AssertEquals_LREAL(
    Expected := 30.0,
    Actual := fbQ1.GetNormSq(),
    Delta := 1e-10,
    Message := 'Norm squared was not the expected value.'
);

AssertEquals_LREAL(
    Expected := 0.047543581616482,
    Actual := fbQ1.GetNormSq(),
    Delta := 1e-10,
    Message := 'Norm squared was not the expected value.'
);

TEST_FINISHED();
END_METHOD


METHOD PRIVATE TestMakeConjExpectCorrectResult
VAR
    fbQ1 : FB_Quaternion;
END_VAR

TEST('TestMakeConjExpectCorrectResult');

fbQ1.Set(1, 2, 3, 4);
fbQ1.MakeConj();

AssertEquals_LREAL(
    Expected := 1,
    Actual := fbQ1.w,
    Delta := 0.0,
    Message := 'Quaternion 1 [w] was not the expected value.'
);

AssertEquals_LREAL(
    Expected := -2,
    Actual := fbQ1.x,
    Delta := 0.0,
    Message := 'Quaternion 1 [x] was not the expected value.'
);

AssertEquals_LREAL(
    Expected := -3,
    Actual := fbQ1.y,
    Delta := 0.0,
    Message := 'Quaternion 1 [y] was not the expected value.'
);

AssertEquals_LREAL(
    Expected := -4,
    Actual := fbQ1.z,
    Delta := 0.0,
    Message := 'Quaternion 1 [z] was not the expected value.'
);

TEST_FINISHED();
END_METHOD


METHOD PRIVATE TestMulQuatExpectCorrectResult
VAR
    fbQ1 : FB_Quaternion;
    fbQ2 : FB_Quaternion;
    fbQ3 : FB_Quaternion;
END_VAR

TEST('TestMulQuatExpectCorrectResult');

fbQ1.Set(1, 2, 3, 4);
fbQ2.Set(0.217115689381933, -0.00950871632329635, 0.01743264659271, -0.00316957210776545);
fbQ3.Set(2, -1, -5, 2);

fbQ1.MulQuat(fbQ2);
fbQ3.MulQuat(fbQ1);

// Q1
AssertEquals_LREAL(
    Expected := 0.196513470681458,
    Actual := fbQ1.w,
    Delta := 1e-10,
    Message := 'Quaternion 1 [w] was not the expected value.'
);

AssertEquals_LREAL(
    Expected := 0.345483359746434,
    Actual := fbQ1.x,
    Delta := 1e-10,
    Message := 'Quaternion 1 [x] was not the expected value.'
);

AssertEquals_LREAL(
    Expected := 0.637083993660856,
    Actual := fbQ1.y,
    Delta := 1e-10,
    Message := 'Quaternion 1 [y] was not the expected value.'
);

AssertEquals_LREAL(
    Expected := 0.928684627575277,
    Actual := fbQ1.z,
    Delta := 1e-10,
    Message := 'Quaternion 1 [z] was not the expected value.'
);

// Q2
AssertEquals_LREAL(
    Expected := 0.217115689381933,
    Actual := fbQ2.w,
    Delta := 0.0,
    Message := 'Quaternion 2 [w] was not the expected value.'
);

AssertEquals_LREAL(
    Expected := -0.00950871632329635,
    Actual := fbQ2.x,
    Delta := 0.0,
    Message := 'Quaternion 2 [x] was not the expected value.'
);

AssertEquals_LREAL(
    Expected := 0.01743264659271,
    Actual := fbQ2.y,
    Delta := 0.0,
    Message := 'Quaternion 2 [y] was not the expected value.'
);

AssertEquals_LREAL(
    Expected := -0.00316957210776545,
    Actual := fbQ2.z,
    Delta := 0.0,
    Message := 'Quaternion 2 [z] was not the expected value.'
);

// Q3
AssertEquals_LREAL(
    Expected := 2.06656101426307,
    Actual := fbQ3.w,
    Delta := 1e-10,
    Message := 'Quaternion 3 [w] was not the expected value.'
);

AssertEquals_LREAL(
    Expected := -5.42313787638669,
    Actual := fbQ3.x,
    Delta := 1e-10,
    Message := 'Quaternion 3 [x] was not the expected value.'
);

AssertEquals_LREAL(
    Expected := 1.91125198098257,
    Actual := fbQ3.y,
    Delta := 1e-10,
    Message := 'Quaternion 3 [y] was not the expected value.'
);

AssertEquals_LREAL(
    Expected := 3.34072900158479,
    Actual := fbQ3.z,
    Delta := 1e-10,
    Message := 'Quaternion 3 [z] was not the expected value.'
);

TEST_FINISHED();
END_METHOD


METHOD PRIVATE TestNormalizeBy0ExpectErrorUnchanged
VAR
    fbQ1 : FB_Quaternion;

    bError : BOOL;
    sErrorMsg : T_MaxString;
END_VAR

TEST('TestNormalizeBy0ExpectErrorUnchanged');

fbQ1.Set(0, 0, 0, 0);
fbQ1.Normalize(
    bError => bError,
    sErrorMsg => sErrorMsg
);

AssertTrue(
    Condition := bError,
    Message := 'Should have had an error on normalize.'
);

AssertFalse(
    Condition := sErrorMsg = '',
    Message := 'Should not have empty error message on normalize.'
);

AssertEquals_LREAL(
    Expected := 0.0,
    Actual := fbQ1.w,
    Delta := 0.0,
    Message := 'Quaternion 1 [w] was not the expected value.'
);

AssertEquals_LREAL(
    Expected := 0.0,
    Actual := fbQ1.x,
    Delta := 0.0,
    Message := 'Quaternion 1 [x] was not the expected value.'
);

AssertEquals_LREAL(
    Expected := 0.0,
    Actual := fbQ1.y,
    Delta := 0.0,
    Message := 'Quaternion 1 [y] was not the expected value.'
);

AssertEquals_LREAL(
    Expected := 0.0,
    Actual := fbQ1.z,
    Delta := 0.0,
    Message := 'Quaternion 1 [z] was not the expected value.'
);

TEST_FINISHED();
END_METHOD


METHOD PRIVATE TestNormalizeExpectCorrectResult
VAR
    fbQ1 : FB_Quaternion;

    bError : BOOL;
    sErrorMsg : T_MaxString;
END_VAR

TEST('TestNormalizeExpectCorrectResult');

fbQ1.Set(0.217115689381933, -0.00950871632329635, 0.01743264659271, -0.00316957210776545);
fbQ1.Normalize(
    bError => bError,
    sErrorMsg => sErrorMsg
);


AssertFalse(
    Condition := bError,
    Message := 'Should not have had an error on normalize.'
);

AssertTrue(
    Condition := sErrorMsg = '',
    Message := 'Should have empty error message on normalize.'
);

AssertEquals_LREAL(
    Expected := 0.995738410181524,
    Actual := fbQ1.w,
    Delta := 1e-10,
    Message := 'Quaternion 1 [w] was not the expected value.'
);

AssertEquals_LREAL(
    Expected := -0.043608981467804,
    Actual := fbQ1.x,
    Delta := 1e-10,
    Message := 'Quaternion 1 [x] was not the expected value.'
);

AssertEquals_LREAL(
    Expected := 0.0799497993576408,
    Actual := fbQ1.y,
    Delta := 1e-10,
    Message := 'Quaternion 1 [y] was not the expected value.'
);

AssertEquals_LREAL(
    Expected := -0.0145363271559347,
    Actual := fbQ1.z,
    Delta := 1e-10,
    Message := 'Quaternion 1 [z] was not the expected value.'
);

TEST_FINISHED();
END_METHOD


METHOD PRIVATE TestSetExpectCorrectResult
VAR
    fbQ1 : FB_Quaternion;
    fbQ2 : FB_Quaternion;
END_VAR

TEST('TestSetExpectCorrectResult');

fbQ1.Set(1, 2, 3, 4);

AssertFalse(
    Condition := fbQ1.EqualsQuat(fbQ2),
    Message := 'Q1 should not register as equal to Q2'
);

fbQ1.Set(0, 0, 0, 0);

AssertTrue(
    Condition := fbQ1.EqualsQuat(fbQ2),
    Message := 'Q1 should register as equal to Q2 after set operation.'
);

TEST_FINISHED();
END_METHOD


METHOD PRIVATE TestToStringExpectCorrectResult
VAR
    fbQ1 : FB_Quaternion;
    sExpected : T_MaxString;
END_VAR

TEST('TestToStringExpectCorrectResult');

fbQ1.Set(1, 2, 3, 4);
sExpected := '1.0 + 2.0i + 3.0j + 4.0k';

AssertTrue(
    Condition := fbQ1.ToString() = sExpected,
    Message := CONCAT('Expected string to be: [',
               CONCAT(sExpected,
               CONCAT('] but string was: [',
               CONCAT(fbQ1.ToString(),
               ']'))))
);

fbQ1.Set(-1, -2, -3, -4);
sExpected := '-1.0 - 2.0i - 3.0j - 4.0k';

AssertTrue(
    Condition := fbQ1.ToString() = sExpected,
    Message := CONCAT('Expected string to be: [',
               CONCAT(sExpected,
               CONCAT('] but string was: [',
               CONCAT(fbQ1.ToString(),
               ']'))))
);

fbQ1.Set(0, 0, 0, 0);
sExpected := '0.0 + 0.0i + 0.0j + 0.0k';

AssertTrue(
    Condition := fbQ1.ToString() = sExpected,
    Message := CONCAT('Expected string to be: [',
               CONCAT(sExpected,
               CONCAT('] but string was: [',
               CONCAT(fbQ1.ToString(),
               ']'))))
);

TEST_FINISHED();
END_METHOD

END_FUNCTION_BLOCK

// ---- Test/FB_QuatRotateVec3Frame_Test.TcPOU

FUNCTION_BLOCK FB_QuatRotateVec3Frame_Test EXTENDS FB_TestSuite


Test0QuatExpectErrorUnchanged();

TestRandInputExpectCorrectResult_1();

TestRandInputExpectCorrectResult_2();

TestRandInputExpectCorrectResult_3();

TestRandInputExpectCorrectResult_4();

TestRandInputExpectCorrectResult_5();


METHOD PRIVATE Test0QuatExpectErrorUnchanged
VAR
    fbQ1 : FB_Quaternion;
    fbV1 : FB_Vec3;

    bError : BOOL;
    sErrorMsg : T_MaxString;
END_VAR

TEST('Test0QuatExpectErrorUnchanged');

fbQ1.Set(0, 0, 0, 0);
fbV1.Set(1, 1, 1);
fbV1 := F_QuatRotateVec3Frame(
    iQuat := fbQ1,
    iVec3 := fbV1,
    bError => bError,
    sErrorMsg => sErrorMsg
);

AssertTrue(
    Condition := bError,
    Message := 'Should have had an error.'
);

AssertFalse(
    Condition := sErrorMsg = '',
    Message := 'Should not have empty error message.'
);

AssertEquals_LREAL(
    Expected := 1,
    Actual := fbV1.x,
    Delta := 0.0,
    Message := 'Vector 1 [x] was not the expected value.'
);

AssertEquals_LREAL(
    Expected := 1,
    Actual := fbV1.y,
    Delta := 0.0,
    Message := 'Vector 1 [y] was not the expected value.'
);

AssertEquals_LREAL(
    Expected := 1,
    Actual := fbV1.z,
    Delta := 0.0,
    Message := 'Vector 1 [z] was not the expected value.'
);

TEST_FINISHED();
END_METHOD


METHOD PRIVATE TestRandInputExpectCorrectResult_1
VAR
    fbQ1 : FB_Quaternion;
    fbV1 : FB_Vec3;

    bError : BOOL;
    sErrorMsg : T_MaxString;
END_VAR

TEST('TestRandInputExpectCorrectResult_1');

fbQ1.Set(0.350952380892271, 0.513249539867053, 0.401808033751942, 0.075966691690842);
fbV1.Set(0.239916153553658, 0.123318934835166, 0.183907788282417);
fbV1 := F_QuatRotateVec3Frame(
    iQuat := fbQ1,
    iVec3 := fbV1,
    bError => bError,
    sErrorMsg => sErrorMsg,
);

AssertFalse(
    Condition := bError,
    Message := 'Should not have had an error.'
);

AssertTrue(
    Condition := sErrorMsg = '',
    Message := 'Should have empty error message.'
);

AssertEquals_LREAL(
    Expected := 0.1309889114846021,
    Actual := fbV1.x,
    Delta := 1e-10,
    Message := 'Vector 1 [x] was not the expected value.'
);

AssertEquals_LREAL(
    Expected := 0.298917056874025,
    Actual := fbV1.y,
    Delta := 1e-10,
    Message := 'Vector 1 [y] was not the expected value.'
);

AssertEquals_LREAL(
    Expected := -0.008938299258921,
    Actual := fbV1.z,
    Delta := 1e-10,
    Message := 'Vector 1 [z] was not the expected value.'
);

TEST_FINISHED();
END_METHOD


METHOD PRIVATE TestRandInputExpectCorrectResult_2
VAR
    fbQ1 : FB_Quaternion;
    fbV1 : FB_Vec3;

    bError : BOOL;
    sErrorMsg : T_MaxString;
END_VAR

TEST('TestRandInputExpectCorrectResult_2');

fbQ1.Set(0.239952525664903, 0.417267069084370, 0.049654430325742, 0.902716109915281);
fbV1.Set(0.944787189721646, 0.490864092468080, 0.489252638400019);
fbV1 := F_QuatRotateVec3Frame(
    iQuat := fbQ1,
    iVec3 := fbV1,
    bError => bError,
    sErrorMsg => sErrorMsg,
);

AssertFalse(
    Condition := bError,
    Message := 'Should not have had an error.'
);

AssertTrue(
    Condition := sErrorMsg = '',
    Message := 'Should have empty error message.'
);

AssertEquals_LREAL(
    Expected := 0.0348639784144761,
    Actual := fbV1.x,
    Delta := 1e-10,
    Message := 'Vector 1 [x] was not the expected value.'
);

AssertEquals_LREAL(
    Expected := -0.652315007988924,
    Actual := fbV1.y,
    Delta := 1e-10,
    Message := 'Vector 1 [y] was not the expected value.'
);

AssertEquals_LREAL(
    Expected := 0.972732321185814,
    Actual := fbV1.z,
    Delta := 1e-10,
    Message := 'Vector 1 [z] was not the expected value.'
);

TEST_FINISHED();
END_METHOD


METHOD PRIVATE TestRandInputExpectCorrectResult_3
VAR
    fbQ1 : FB_Quaternion;
    fbV1 : FB_Vec3;

    bError : BOOL;
    sErrorMsg : T_MaxString;
END_VAR

TEST('TestRandInputExpectCorrectResult_3');

fbQ1.Set(0.337719409821377, 0.900053846417662, 0.369246781120215, 0.111202755293787);
fbV1.Set(0.780252068321138, 0.389738836961253, 0.241691285913833);
fbV1 := F_QuatRotateVec3Frame(
    iQuat := fbQ1,
    iVec3 := fbV1,
    bError => bError,
    sErrorMsg => sErrorMsg,
);

AssertFalse(
    Condition := bError,
    Message := 'Should not have had an error.'
);

AssertTrue(
    Condition := sErrorMsg = '',
    Message := 'Should have empty error message.'
);

AssertEquals_LREAL(
    Expected := 0.8216066116511471,
    Actual := fbV1.x,
    Delta := 1e-10,
    Message := 'Vector 1 [x] was not the expected value.'
);

AssertEquals_LREAL(
    Expected := 0.376413959087926,
    Actual := fbV1.y,
    Delta := 1e-10,
    Message := 'Vector 1 [y] was not the expected value.'
);

AssertEquals_LREAL(
    Expected := -0.048779462244682,
    Actual := fbV1.z,
    Delta := 1e-10,
    Message := 'Vector 1 [z] was not the expected value.'
);

TEST_FINISHED();
END_METHOD


METHOD PRIVATE TestRandInputExpectCorrectResult_4
VAR
    fbQ1 : FB_Quaternion;
    fbV1 : FB_Vec3;

    bError : BOOL;
    sErrorMsg : T_MaxString;
END_VAR

TEST('TestRandInputExpectCorrectResult_4');

fbQ1.Set(0.403912145588115, 0.096454525168389, 0.131973292606335, 0.942050590775485);
fbV1.Set(0.956134540229802, 0.575208595078466, 0.059779542947156);
fbV1 := F_QuatRotateVec3Frame(
    iQuat := fbQ1,
    iVec3 := fbV1,
    bError => bError,
    sErrorMsg => sErrorMsg,
);

AssertFalse(
    Condition := bError,
    Message := 'Should not have had an error.'
);

AssertTrue(
    Condition := sErrorMsg = '',
    Message := 'Should have empty error message.'
);

AssertEquals_LREAL(
    Expected := -0.2259527588901821,
    Actual := fbV1.x,
    Delta := 1e-10,
    Message := 'Vector 1 [x] was not the expected value.'
);

AssertEquals_LREAL(
    Expected := -1.017084075917310,
    Actual := fbV1.y,
    Delta := 1e-10,
    Message := 'Vector 1 [y] was not the expected value.'
);

AssertEquals_LREAL(
    Expected := 0.403877597661613,
    Actual := fbV1.z,
    Delta := 1e-10,
    Message := 'Vector 1 [z] was not the expected value.'
);

TEST_FINISHED();
END_METHOD


METHOD PRIVATE TestRandInputExpectCorrectResult_5
VAR
    fbQ1 : FB_Quaternion;
    fbV1 : FB_Vec3;

    bError : BOOL;
    sErrorMsg : T_MaxString;
END_VAR

TEST('TestRandInputExpectCorrectResult_5');

fbQ1.Set(0.234779913372406, 0.353158571222071, 0.821194040197959, 0.015403437651555);
fbV1.Set(0.043023801657808, 0.168990029462704, 0.649115474956452);
fbV1 := F_QuatRotateVec3Frame(
    iQuat := fbQ1,
    iVec3 := fbV1,
    bError => bError,
    sErrorMsg => sErrorMsg,
);

AssertFalse(
    Condition := bError,
    Message := 'Should not have had an error.'
);

AssertTrue(
    Condition := sErrorMsg = '',
    Message := 'Should have empty error message.'
);

AssertEquals_LREAL(
    Expected := -0.1934394675708541,
    Actual := fbV1.x,
    Delta := 1e-10,
    Message := 'Vector 1 [x] was not the expected value.'
);

AssertEquals_LREAL(
    Expected := 0.293602775485964,
    Actual := fbV1.y,
    Delta := 1e-10,
    Message := 'Vector 1 [y] was not the expected value.'
);

AssertEquals_LREAL(
    Expected := -0.572833448750751,
    Actual := fbV1.z,
    Delta := 1e-10,
    Message := 'Vector 1 [z] was not the expected value.'
);

TEST_FINISHED();
END_METHOD

END_FUNCTION_BLOCK

// ---- Test/FB_QuatRotateVec3Point_Test.TcPOU

FUNCTION_BLOCK FB_QuatRotateVec3Point_Test EXTENDS FB_TestSuite


Test0QuatExpectErrorUnchanged();

TestRandInputExpectCorrectResult_1();

TestRandInputExpectCorrectResult_2();

TestRandInputExpectCorrectResult_3();

TestRandInputExpectCorrectResult_4();

TestRandInputExpectCorrectResult_5();


METHOD PRIVATE Test0QuatExpectErrorUnchanged
VAR
    fbQ1 : FB_Quaternion;
    fbV1 : FB_Vec3;

    bError : BOOL;
    sErrorMsg : T_MaxString;
END_VAR

TEST('Test0QuatExpectErrorUnchanged');

fbQ1.Set(0, 0, 0, 0);
fbV1.Set(1, 1, 1);
fbV1 := F_QuatRotateVec3Point(
    iQuat := fbQ1,
    iVec3 := fbV1,
    bError => bError,
    sErrorMsg => sErrorMsg
);

AssertTrue(
    Condition := bError,
    Message := 'Should have had an error.'
);

AssertFalse(
    Condition := sErrorMsg = '',
    Message := 'Should not have empty error message.'
);

AssertEquals_LREAL(
    Expected := 1,
    Actual := fbV1.x,
    Delta := 0.0,
    Message := 'Vector 1 [x] was not the expected value.'
);

AssertEquals_LREAL(
    Expected := 1,
    Actual := fbV1.y,
    Delta := 0.0,
    Message := 'Vector 1 [y] was not the expected value.'
);

AssertEquals_LREAL(
    Expected := 1,
    Actual := fbV1.z,
    Delta := 0.0,
    Message := 'Vector 1 [z] was not the expected value.'
);

TEST_FINISHED();
END_METHOD


METHOD PRIVATE TestRandInputExpectCorrectResult_1
VAR
    fbQ1 : FB_Quaternion;
    fbV1 : FB_Vec3;

    bError : BOOL;
    sErrorMsg : T_MaxString;
END_VAR

TEST('TestRandInputExpectCorrectResult_1');

fbQ1.Set(0.731722385658670, 0.647745963136307, 0.450923706430945, 0.547008892286345);
fbV1.Set(0.296320805607773, 0.744692807074156, 0.188955015032545);
fbV1 := F_QuatRotateVec3Point(
    iQuat := fbQ1,
    iVec3 := fbV1,
    bError => bError,
    sErrorMsg => sErrorMsg,
);

AssertFalse(
    Condition := bError,
    Message := 'Should not have had an error.'
);

AssertTrue(
    Condition := sErrorMsg = '',
    Message := 'Should have empty error message.'
);

AssertEquals_LREAL(
    Expected := 0.1588618332623411,
    Actual := fbV1.x,
    Delta := 1e-10,
    Message := 'Vector 1 [x] was not the expected value.'
);

AssertEquals_LREAL(
    Expected := 0.232767876109413,
    Actual := fbV1.y,
    Delta := 1e-10,
    Message := 'Vector 1 [y] was not the expected value.'
);

AssertEquals_LREAL(
    Expected := 0.773730849995020,
    Actual := fbV1.z,
    Delta := 1e-10,
    Message := 'Vector 1 [z] was not the expected value.'
);

TEST_FINISHED();
END_METHOD


METHOD PRIVATE TestRandInputExpectCorrectResult_2
VAR
    fbQ1 : FB_Quaternion;
    fbV1 : FB_Vec3;

    bError : BOOL;
    sErrorMsg : T_MaxString;
END_VAR

TEST('TestRandInputExpectCorrectResult_2');

fbQ1.Set(0.686775433365315, 0.183511155737270, 0.368484596490336, 0.625618560729690);
fbV1.Set(0.780227435151377, 0.081125768865785, 0.929385970968730);
fbV1 := F_QuatRotateVec3Point(
    iQuat := fbQ1,
    iVec3 := fbV1,
    bError => bError,
    sErrorMsg => sErrorMsg,
);

AssertFalse(
    Condition := bError,
    Message := 'Should not have had an error.'
);

AssertTrue(
    Condition := sErrorMsg = '',
    Message := 'Should have empty error message.'
);

AssertEquals_LREAL(
    Expected := 0.5888629779440591,
    Actual := fbV1.x,
    Delta := 1e-10,
    Message := 'Vector 1 [x] was not the expected value.'
);

AssertEquals_LREAL(
    Expected := 0.953999228289107,
    Actual := fbV1.y,
    Delta := 1e-10,
    Message := 'Vector 1 [y] was not the expected value.'
);

AssertEquals_LREAL(
    Expected := 0.471402576998784,
    Actual := fbV1.z,
    Delta := 1e-10,
    Message := 'Vector 1 [z] was not the expected value.'
);

TEST_FINISHED();
END_METHOD


METHOD PRIVATE TestRandInputExpectCorrectResult_3
VAR
    fbQ1 : FB_Quaternion;
    fbV1 : FB_Vec3;

    bError : BOOL;
    sErrorMsg : T_MaxString;
END_VAR

TEST('TestRandInputExpectCorrectResult_3');

fbQ1.Set(0.775712678608402, 0.486791632403172, 0.435858588580919, 0.446783749429806);
fbV1.Set(0.306349472016557, 0.508508655381127, 0.510771564172110);
fbV1 := F_QuatRotateVec3Point(
    iQuat := fbQ1,
    iVec3 := fbV1,
    bError => bError,
    sErrorMsg => sErrorMsg,
);

AssertFalse(
    Condition := bError,
    Message := 'Should not have had an error.'
);

AssertTrue(
    Condition := sErrorMsg = '',
    Message := 'Should have empty error message.'
);

AssertEquals_LREAL(
    Expected := 0.4628031823996781,
    Actual := fbV1.x,
    Delta := 1e-10,
    Message := 'Vector 1 [x] was not the expected value.'
);

AssertEquals_LREAL(
    Expected := 0.273642504441062,
    Actual := fbV1.y,
    Delta := 1e-10,
    Message := 'Vector 1 [y] was not the expected value.'
);

AssertEquals_LREAL(
    Expected := 0.569430976056908,
    Actual := fbV1.z,
    Delta := 1e-10,
    Message := 'Vector 1 [z] was not the expected value.'
);

TEST_FINISHED();
END_METHOD


METHOD PRIVATE TestRandInputExpectCorrectResult_4
VAR
    fbQ1 : FB_Quaternion;
    fbV1 : FB_Vec3;

    bError : BOOL;
    sErrorMsg : T_MaxString;
END_VAR

TEST('TestRandInputExpectCorrectResult_4');

fbQ1.Set(0.817627708322262, 0.794831416883453, 0.644318130193692, 0.378609382660268);
fbV1.Set(0.811580458282477, 0.532825588799455, 0.350727103576883);
fbV1 := F_QuatRotateVec3Point(
    iQuat := fbQ1,
    iVec3 := fbV1,
    bError => bError,
    sErrorMsg => sErrorMsg,
);

AssertFalse(
    Condition := bError,
    Message := 'Should not have had an error.'
);

AssertTrue(
    Condition := sErrorMsg = '',
    Message := 'Should have empty error message.'
);

AssertEquals_LREAL(
    Expected := 0.7523821769332431,
    Actual := fbV1.x,
    Delta := 1e-10,
    Message := 'Vector 1 [x] was not the expected value.'
);

AssertEquals_LREAL(
    Expected := 0.652796600025488,
    Actual := fbV1.y,
    Delta := 1e-10,
    Message := 'Vector 1 [y] was not the expected value.'
);

AssertEquals_LREAL(
    Expected := 0.270837789751114,
    Actual := fbV1.z,
    Delta := 1e-10,
    Message := 'Vector 1 [z] was not the expected value.'
);

TEST_FINISHED();
END_METHOD


METHOD PRIVATE TestRandInputExpectCorrectResult_5
VAR
    fbQ1 : FB_Quaternion;
    fbV1 : FB_Vec3;

    bError : BOOL;
    sErrorMsg : T_MaxString;
END_VAR

TEST('TestRandInputExpectCorrectResult_5');

fbQ1.Set(0.939001561999887, 0.875942811492984, 0.550156342898422, 0.622475086001227);
fbV1.Set(0.587044704531417, 0.207742292733028, 0.301246330279491);
fbV1 := F_QuatRotateVec3Point(
    iQuat := fbQ1,
    iVec3 := fbV1,
    bError => bError,
    sErrorMsg => sErrorMsg,
);

AssertFalse(
    Condition := bError,
    Message := 'Should not have had an error.'
);

AssertTrue(
    Condition := sErrorMsg = '',
    Message := 'Should have empty error message.'
);

AssertEquals_LREAL(
    Expected := 0.4959148487251781,
    Actual := fbV1.x,
    Delta := 1e-10,
    Message := 'Vector 1 [x] was not the expected value.'
);

AssertEquals_LREAL(
    Expected := 0.414249906357875,
    Actual := fbV1.y,
    Delta := 1e-10,
    Message := 'Vector 1 [y] was not the expected value.'
);

AssertEquals_LREAL(
    Expected := 0.246967962925536,
    Actual := fbV1.z,
    Delta := 1e-10,
    Message := 'Vector 1 [z] was not the expected value.'
);

TEST_FINISHED();
END_METHOD

END_FUNCTION_BLOCK

// ---- Test/FB_Vec3_Test.TcPOU

FUNCTION_BLOCK FB_Vec3_Test EXTENDS FB_TestSuite


TestAddVec3ExpectCorrectResult();

TestCrossVec3ExpectCorrectResult();

TestDivScalarBy0ExpectErrorUnchanged();

TestDivScalarExpectNoErrorCorrectResult();

TestDotVec3ExpectCorrectResult();

TestEqualsVec3ExpectCorrectResult();

TestGetNormExpectCorrectResult();

TestGetNormSqExpectCorrectResult();

TestNormalizeBy0ExpectErrorUnchanged();

TestNormalizeExpectCorrectResult();

TestSetExpectCorrectResult();

TestToStringExpectCorrectResult();


METHOD PRIVATE TestAddVec3ExpectCorrectResult
VAR
    fbV1 : FB_Vec3;
    fbV2 : FB_Vec3;
    fbV3 : FB_Vec3;
END_VAR

TEST('TestAddVec3ExpectCorrectResult');

fbV1.Set(1, 2, 3);
fbV2.Set(5, 11, 14);
fbV3.Set(2, -1, -5);

fbV1.AddVec3(fbV2);
fbV3.AddVec3(fbV1);

// V1
AssertEquals_LREAL(
    Expected := 6.0,
    Actual := fbV1.x,
    Delta := 0.0,
    Message := 'Vector 1 [x] was not the expected value.'
);

AssertEquals_LREAL(
    Expected := 13.0,
    Actual := fbV1.y,
    Delta := 0.0,
    Message := 'Vector 1 [y] was not the expected value.'
);

AssertEquals_LREAL(
    Expected := 17.0,
    Actual := fbV1.z,
    Delta := 0.0,
    Message := 'Vector 1 [z] was not the expected value.'
);

// V2
AssertEquals_LREAL(
    Expected := 5.0,
    Actual := fbV2.x,
    Delta := 0.0,
    Message := 'Vector 2 [x] was not the expected value.'
);

AssertEquals_LREAL(
    Expected := 11.0,
    Actual := fbV2.y,
    Delta := 0.0,
    Message := 'Vector 2 [y] was not the expected value.'
);

AssertEquals_LREAL(
    Expected := 14.0,
    Actual := fbV2.z,
    Delta := 0.0,
    Message := 'Vector 2 [z] was not the expected value.'
);

// V3
AssertEquals_LREAL(
    Expected := 8.0,
    Actual := fbV3.x,
    Delta := 0.0,
    Message := 'Vector 3 [x] was not the expected value.'
);

AssertEquals_LREAL(
    Expected := 12.0,
    Actual := fbV3.y,
    Delta := 0.0,
    Message := 'Vector 3 [y] was not the expected value.'
);

AssertEquals_LREAL(
    Expected := 12.0,
    Actual := fbV3.z,
    Delta := 0.0,
    Message := 'Vector 3 [z] was not the expected value.'
);

TEST_FINISHED();
END_METHOD


METHOD PRIVATE TestCrossVec3ExpectCorrectResult
VAR
    fbV1 : FB_Vec3;
    fbV2 : FB_Vec3;
    fbV3 : FB_Vec3;
END_VAR

TEST('TestCrossVec3ExpectCorrectResult');

fbV1.Set(1, 2, 3);
fbV2.Set(0.217115689381933, -0.00950871632329635, 0.01743264659271);
fbV3.Set(2, -1, -5);

fbV1.CrossVec3(fbV2);
fbV3.CrossVec3(fbV1);

// V1
AssertEquals_LREAL(
    Expected := 0.063391442155309,
    Actual := fbV1.x,
    Delta := 1e-10,
    Message := 'Vector 1 [x] was not the expected value.'
);

AssertEquals_LREAL(
    Expected := 0.633914421553089,
    Actual := fbV1.y,
    Delta := 1e-10,
    Message := 'Vector 1 [y] was not the expected value.'
);

AssertEquals_LREAL(
    Expected := -0.443740095087162,
    Actual := fbV1.z,
    Delta := 1e-10,
    Message := 'Vector 1 [z] was not the expected value.'
);

// V2
AssertEquals_LREAL(
    Expected := 0.217115689381933,
    Actual := fbV2.x,
    Delta := 0.0,
    Message := 'Vector 2 [x] was not the expected value.'
);

AssertEquals_LREAL(
    Expected := -0.00950871632329635,
    Actual := fbV2.y,
    Delta := 0.0,
    Message := 'Vector 2 [y] was not the expected value.'
);

AssertEquals_LREAL(
    Expected := 0.01743264659271,
    Actual := fbV2.z,
    Delta := 0.0,
    Message := 'Vector 2 [z] was not the expected value.'
);

// V3
AssertEquals_LREAL(
    Expected := 3.613312202852607,
    Actual := fbV3.x,
    Delta := 1e-10,
    Message := 'Vector 3 [x] was not the expected value.'
);

AssertEquals_LREAL(
    Expected := 0.570522979397780,
    Actual := fbV3.y,
    Delta := 1e-10,
    Message := 'Vector 3 [y] was not the expected value.'
);

AssertEquals_LREAL(
    Expected := 1.331220285261487,
    Actual := fbV3.z,
    Delta := 1e-10,
    Message := 'Vector 3 [z] was not the expected value.'
);

TEST_FINISHED();
END_METHOD


METHOD PRIVATE TestDivScalarBy0ExpectErrorUnchanged
VAR
    fbV1 : FB_Vec3;

    bError : BOOL;
    sErrorMsg : T_MaxString;
END_VAR

TEST('TestDivScalarBy0ExpectErrorUnchanged');

fbV1.Set(1, 2, 3);

fbV1.DivScalar(
    fScalar := 0.0,
    bError => bError,
    sErrorMsg => sErrorMsg
);

AssertTrue(
    Condition := bError,
    Message := 'Should have had an error on the scalar division operation.'
);

AssertFalse(
    Condition := sErrorMsg = '',
    Message := 'Should not have had an empty error message on the scalar division operation.'
);

// V1
AssertEquals_LREAL(
    Expected := 1,
    Actual := fbV1.x,
    Delta := 1e-10,
    Message := 'Vector 1 [x] was not the expected value.'
);

AssertEquals_LREAL(
    Expected := 2,
    Actual := fbV1.y,
    Delta := 1e-10,
    Message := 'Vector 1 [y] was not the expected value.'
);

AssertEquals_LREAL(
    Expected := 3,
    Actual := fbV1.z,
    Delta := 1e-10,
    Message := 'Vector 1 [z] was not the expected value.'
);

TEST_FINISHED();
END_METHOD


METHOD PRIVATE TestDivScalarExpectNoErrorCorrectResult
VAR
    fbV1 : FB_Vec3;

    bError : BOOL;
    sErrorMsg : T_MaxString;
END_VAR

TEST('TestDivScalarExpectNoErrorCorrectResult');

fbV1.Set(1, 2, 3);

fbV1.DivScalar(
    fScalar := 2.0,
    bError => bError,
    sErrorMsg => sErrorMsg
);

AssertFalse(
    Condition := bError,
    Message := 'Should not have had an error on the scalar division operation.'
);

AssertTrue(
    Condition := sErrorMsg = '',
    Message := 'Should have had an empty error message on the scalar division operation.'
);

// V1
AssertEquals_LREAL(
    Expected := 0.5,
    Actual := fbV1.x,
    Delta := 1e-10,
    Message := 'Vector 1 [x] was not the expected value.'
);

AssertEquals_LREAL(
    Expected := 1.0,
    Actual := fbV1.y,
    Delta := 1e-10,
    Message := 'Vector 1 [y] was not the expected value.'
);

AssertEquals_LREAL(
    Expected := 1.5,
    Actual := fbV1.z,
    Delta := 1e-10,
    Message := 'Vector 1 [z] was not the expected value.'
);

TEST_FINISHED();
END_METHOD


METHOD PRIVATE TestDotVec3ExpectCorrectResult
VAR
    fbV1 : FB_Vec3;
    fbV2 : FB_Vec3;
    fbV3 : FB_Vec3;
END_VAR

TEST('TestDotVec3ExpectCorrectResult');

fbV1.Set(1, 2, 3);
fbV2.Set(0.217115689381933, -0.00950871632329635, 0.01743264659271);
fbV3.Set(43, 12, 856);

AssertEquals_LREAL(
    Expected := 0.250396196513470,
    Actual := fbV1.DotVec3(fbV2),
    Delta := 1e-10,
    Message := 'Dot product was not the expected value.'
);

AssertEquals_LREAL(
    Expected := 24.144215530903324,
    Actual := fbV2.DotVec3(fbV3),
    Delta := 1e-10,
    Message := 'Dot product was not the expected value.'
);

TEST_FINISHED();
END_METHOD


METHOD PRIVATE TestEqualsVec3ExpectCorrectResult
VAR
    fbV1 : FB_Vec3;
    fbV2 : FB_Vec3;
    fbV3 : FB_Vec3;
END_VAR

TEST('TestEqualsVec3ExpectCorrectResult');

fbV1.Set(1, 2, 3);
fbV2.Set(5, 11, 14);
fbV3.Set(1, 2, 3);

AssertTrue(
    Condition := fbV1.EqualsVec3(fbV3),
    Message := 'V1 should register as equal to V3'
);

AssertTrue(
    Condition := fbV3.EqualsVec3(fbV1),
    Message := 'V3 should register as equal to V1'
);

AssertFalse(
    Condition := fbV1.EqualsVec3(fbV2),
    Message := 'V1 should not register as equal to V2'
);

AssertFalse(
    Condition := fbV2.EqualsVec3(fbV1),
    Message := 'V2 should not register as equal to V1'
);

TEST_FINISHED();
END_METHOD


METHOD PRIVATE TestGetNormExpectCorrectResult
VAR
    fbV1 : FB_Vec3;
    fbV2 : FB_Vec3;
END_VAR

TEST('TestGetNormExpectCorrectResult');

fbV1.Set(1, 2, 3);
fbV2.Set(0.217115689381933, -0.00950871632329635, 0.01743264659271);

AssertEquals_LREAL(
    Expected := 3.741657386773941,
    Actual := fbV1.GetNorm(),
    Delta := 1e-10,
    Message := 'Norm was not the expected value.'
);

AssertEquals_LREAL(
    Expected := 0.218021869153384,
    Actual := fbV2.GetNorm(),
    Delta := 1e-10,
    Message := 'Norm was not the expected value.'
);

TEST_FINISHED();
END_METHOD


METHOD PRIVATE TestGetNormSqExpectCorrectResult
VAR
    fbV1 : FB_Vec3;
    fbV2 : FB_Vec3;
END_VAR

TEST('TestGetNormSqExpectCorrectResult');

fbV1.Set(1, 2, 3);
fbV2.Set(0.217115689381933, -0.00950871632329635, 0.01743264659271);

AssertEquals_LREAL(
    Expected := 14.0,
    Actual := fbV1.GetNormSq(),
    Delta := 1e-10,
    Message := 'Norm squared was not the expected value.'
);

AssertEquals_LREAL(
    Expected := 0.047533535429135,
    Actual := fbV2.GetNormSq(),
    Delta := 1e-10,
    Message := 'Norm squared was not the expected value.'
);

TEST_FINISHED();
END_METHOD


METHOD PRIVATE TestNormalizeBy0ExpectErrorUnchanged
VAR
    fbV1 : FB_Vec3;

    bError : BOOL;
    sErrorMsg : T_MaxString;
END_VAR

TEST('TestNormalizeBy0ExpectErrorUnchanged');

fbV1.Set(0, 0, 0);
fbV1.Normalize(
    bError => bError,
    sErrorMsg => sErrorMsg
);

AssertTrue(
    Condition := bError,
    Message := 'Should have had an error on normalize.'
);

AssertFalse(
    Condition := sErrorMsg = '',
    Message := 'Should not have empty error message on normalize.'
);

AssertEquals_LREAL(
    Expected := 0.0,
    Actual := fbV1.x,
    Delta := 0.0,
    Message := 'Vector 1 [x] was not the expected value.'
);

AssertEquals_LREAL(
    Expected := 0.0,
    Actual := fbV1.y,
    Delta := 0.0,
    Message := 'Vector 1 [y] was not the expected value.'
);

AssertEquals_LREAL(
    Expected := 0.0,
    Actual := fbV1.z,
    Delta := 0.0,
    Message := 'Vector 1 [z] was not the expected value.'
);

TEST_FINISHED();
END_METHOD


METHOD PRIVATE TestNormalizeExpectCorrectResult
VAR
    fbV1 : FB_Vec3;

    bError : BOOL;
    sErrorMsg : T_MaxString;
END_VAR

TEST('TestNormalizeExpectCorrectResult');

fbV1.Set(0.217115689381933, -0.00950871632329635, 0.01743264659271);
fbV1.Normalize(
    bError => bError,
    sErrorMsg => sErrorMsg
);

AssertFalse(
    Condition := bError,
    Message := 'Should not have had an error on normalize.'
);

AssertTrue(
    Condition := sErrorMsg = '',
    Message := 'Should have empty error message on normalize.'
);

AssertEquals_LREAL(
    Expected := 0.995843629013136,
    Actual := fbV1.x,
    Delta := 1e-10,
    Message := 'Vector 1 [x] was not the expected value.'
);

AssertEquals_LREAL(
    Expected := -0.043613589591816,
    Actual := fbV1.y,
    Delta := 1e-10,
    Message := 'Vector 1 [y] was not the expected value.'
);

AssertEquals_LREAL(
    Expected := 0.079958247584997,
    Actual := fbV1.z,
    Delta := 1e-10,
    Message := 'Vector 1 [z] was not the expected value.'
);

TEST_FINISHED();
END_METHOD


METHOD PRIVATE TestSetExpectCorrectResult
VAR
    fbV1 : FB_Vec3;
    fbV2 : FB_Vec3;
END_VAR

TEST('TestSetExpectCorrectResult');

fbV1.Set(1, 2, 3);

AssertFalse(
    Condition := fbV1.EqualsVec3(fbV2),
    Message := 'V1 should not register as equal to V2'
);

fbV1.Set(0, 0, 0);

AssertTrue(
    Condition := fbV1.EqualsVec3(fbV2),
    Message := 'V1 should register as equal to V2 after set operation.'
);

TEST_FINISHED();
END_METHOD


METHOD PRIVATE TestToStringExpectCorrectResult
VAR
    fbV1 : FB_Vec3;
    sExpected : T_MaxString;
END_VAR

TEST('TestToStringExpectCorrectResult');

fbV1.Set(1, 2, 3);
sExpected := '(1.0, 2.0, 3.0)';

AssertTrue(
    Condition := fbV1.ToString() = sExpected,
    Message := CONCAT('Expected string to be: [',
               CONCAT(sExpected,
               CONCAT('] but string was: [',
               CONCAT(fbV1.ToString(),
               ']'))))
);

fbV1.Set(-1, -2, -3);
sExpected := '(-1.0, -2.0, -3.0)';

AssertTrue(
    Condition := fbV1.ToString() = sExpected,
    Message := CONCAT('Expected string to be: [',
               CONCAT(sExpected,
               CONCAT('] but string was: [',
               CONCAT(fbV1.ToString(),
               ']'))))
);

fbV1.Set(0, 0, 0);
sExpected := '(0.0, 0.0, 0.0)';

AssertTrue(
    Condition := fbV1.ToString() = sExpected,
    Message := CONCAT('Expected string to be: [',
               CONCAT(sExpected,
               CONCAT('] but string was: [',
               CONCAT(fbV1.ToString(),
               ']'))))
);

TEST_FINISHED();
END_METHOD

END_FUNCTION_BLOCK
